{attribute 'linkalways'} 
{attribute 'no_explicit_call' := 'This FB is a CLASS and must be accessed using methods or properties'}
{attribute 'enable_dynamic_creation'}
FUNCTION_BLOCK Node_ContainerType_Vector_TcVnPoint2_DINT EXTENDS Node
VAR
    out : _GUID;
END_VAR

METHOD PUBLIC  Clone : I_Node
VAR
	pNode : POINTER TO Node_ContainerType_Vector_TcVnPoint2_DINT;
END_VAR
pNode := __NEW(Node_ContainerType_Vector_TcVnPoint2_DINT);
Clone := pNode^;
END_METHOD

METHOD FB_init : BOOL
VAR_INPUT
	bInitRetains : BOOL; // if TRUE, the retain variables are initialized (warm start / cold start)
	bInCopyCode : BOOL;  // if TRUE, the instance afterwards gets moved into the copy code (online change)
END_VAR
AddOutput('out', out);
END_METHOD

METHOD PROTECTED OnExecute
out.Value := ContainerType_Vector_TcVnPoint2_DINT;
END_METHOD

END_FUNCTION_BLOCK

(* stored: Version 1.1.0.1, ProductVersion 3.1.4026.17
   POU Node_ContainerType_Vector_TcVnPoint2_DINT: Id {91004355-4254-0445-032e-de0e12fb9d84}, SpecialFunc None
   Folder Constructor: Id {4e8535ba-9c67-04f9-33f2-d4ccef9b0264}
   Method Clone: Id {2dbef042-27ee-0ffc-0a1f-82f65bb015af}
   Method FB_init: Id {798b156f-3894-0490-2cd4-0a870063095f}
   Method OnExecute: Id {7d171fb8-f66a-0d87-0969-8969eb48739d} *)
